TYPE ST_FIO_AxisIO :
STRUCT
    SetPos : LREAL;   // output: position command to "analog output"
    ActPos : LREAL;   // input: feedback from "analog input"
END_STRUCT
END_TYPE

(* stored: Version 1.1.0.1
   DUT ST_FIO_AxisIO: Id {ae82dc49-1a08-4dfe-b557-7faee9b5f922} *)
